// TIA Portal V19 export
VAR_GLOBAL   // PLC tag table "Safety_IO"
   IS_EstopLeftRopePull AT %I500.1 : Bool;   // Right e-stop rope pull switch - Channel 1   {ExternalAccessible false}
   IS_EstopRightRopePull AT %I500.0 : Bool;   // Left e-stop rope pull switch - Channel 1   {ExternalAccessible false}
   IS_EStopMainCabinet AT %I500.2 : Bool;   // Main panel e-stop - Channel 1   {ExternalAccessible false}
   IS_EStopEntryDoor AT %I500.3 : Bool;   // Entry door e-stop - Channel 1   {ExternalAccessible false}
   IS_EstopLeftRopePull_Ch2 AT %I500.5 : Bool;   // Right e-stop rope pull switch - Channel 2   {ExternalAccessible false}
   IS_EstopRightRopePull_Ch2 AT %I500.4 : Bool;   // Left e-stop rope pull switch - Channel 2   {ExternalAccessible false}
   IS_EStopMainCabinet_Ch2 AT %I500.6 : Bool;   // Main panel e-stop - Channel 2   {ExternalAccessible false}
   IS_EStopEntryDoor_Ch2 AT %I500.7 : Bool;   // Entry door e-stop - Channel 2   {ExternalAccessible false}
   IS_DoorAcces_Ch1 AT %I507.0 : Bool;   // Door acces state - Channel 1   {ExternalAccessible false}
   IS_GateAccesCBS AT %I507.1 : Bool;   // CBS Gate Acces State - Channel 1   {ExternalAccessible false}
   IS_EStopControlRoom AT %I507.2 : Bool;   // Control Room E-Stop - Channel 1   {ExternalAccessible false}
   IS_DoorAcces_Ch2 AT %I507.4 : Bool;   // Door acces state - Channel 2   {ExternalAccessible false}
   IS_GateAccesCBS_Ch2 AT %I507.5 : Bool;   // CBS Gate Acces State - Channel 2   {ExternalAccessible false}
   IS_EStopControlRoom_Ch2 AT %I507.6 : Bool;   // Control Room E-Stop - Channel 2   {ExternalAccessible false}
   OS_EStopSuctionUnit AT %Q522.1 : Bool;   // E-Stop Suction Unit   {ExternalAccessible false}
   OS_EnableAirSupplyLeftRobot AT %Q522.2 : Bool;   // Air supply robot 1 Ok   {ExternalAccessible false}
   OS_EnableAirSupplyRightRobot AT %Q522.3 : Bool;   // Air supply robot 2 Ok   {ExternalAccessible false}
   OS_EnableAirSupplySuctionUnit AT %Q522.4 : Bool;   // Air supply suction unit Ok   {ExternalAccessible false}
   ISS_EStopSuctionUnit AT %I522.1 : Bool;   // State E-Stop Suction Unit   {ExternalAccessible false}
   ISS_EnableAirSupplyLeftRobot AT %I522.2 : Bool;   // State Air supply robot 1 Ok   {ExternalAccessible false}
   ISS_EnableAirSupplyRightRobot AT %I522.3 : Bool;   // State Air supply robot 2 Ok   {ExternalAccessible false}
   ISS_EnableAirSupplySuctionUnit AT %I522.4 : Bool;   // Air supply suction unit Ok   {ExternalAccessible false}
   ISS_EstopLeftRopePull AT %I501.1 : Bool;   // State Right e-stop rope pull switch - Channel 1   {ExternalAccessible false}
   ISS_EstopRightRopePull AT %I501.0 : Bool;   // State Left e-stop rope pull switch - Channel 1   {ExternalAccessible false}
   ISS_EStopMainCabinet AT %I501.2 : Bool;   // State Main panel e-stop - Channel 1   {ExternalAccessible false}
   ISS_EStopEntryDoor AT %I501.3 : Bool;   // State Entry door e-stop - Channel 1   {ExternalAccessible false}
   ISS_DoorAcces_Ch1 AT %I508.0 : Bool;   // State Door acces state - Channel 1   {ExternalAccessible false}
   ISS_GateAccesCBS AT %I508.1 : Bool;   // State CBS Gate Acces State - Channel 1   {ExternalAccessible false}
   ISS_EStopControlRoom AT %I508.2 : Bool;   // State Control Room E-Stop - Channel 1   {ExternalAccessible false}
   ISS_DoorAcces_Ch2 AT %I508.4 : Bool;   // State Door acces state - Channel 2   {ExternalAccessible false}
   ISB_500 AT %IB500 : SInt;   //    {ExternalWritable false}
   ISB_507 AT %IB507 : SInt;   //    {ExternalWritable false}
   ISB_514 AT %IB514 : SInt;   //    {ExternalWritable false}
   OSB_522 AT %QB522 : SInt;   //    {ExternalWritable false}
   IS_PedestrialDoor AT %I507.3 : Bool;   // Pedestral door acces control   {ExternalAccessible false}
   IS_CaptiveKeyState AT %I514.0 : Bool;   // Captive key in lock - Channel 1   {ExternalAccessible false}
   IS_CaptiveKeyState_Ch2 AT %I514.4 : Bool;   // Captive key in lock - Channel 2   {ExternalAccessible false}
   ISS_CaptiveKeyState AT %I515.0 : Bool;   // State Captive key in lock   {ExternalAccessible false}
   IS_VacuumPumpRunning AT %I507.7 : Bool;   // Vacuum pump runing, zero speed detection   {ExternalAccessible false}
END_VAR
